// Converts all alphabetic characters in a string uppercase characters
FUNCTION F_TOUPPER
VAR_INPUT
	sValue : REFERENCE TO STRING; // String of any size
END_VAR
VAR
	i : T_Size;
END_VAR

WHILE sValue[i] <> 0 DO 
	IF sValue[i] >= 97 AND sValue[i]<= 122 THEN sValue[i] := sValue[i] - 32; END_IF
	i := i + 1;
	END_WHILE

END_FUNCTION

(* stored: Version 1.1.0.1, ProductVersion 3.1.4024.4
   POU F_TOUPPER: Id {f6d5a607-3f58-4a60-959f-aa50bc9b18aa}, SpecialFunc None *)
